// TIA Portal project "Project1" (V14)

(* hardware
DEVICE "S71500/ET200MP station_1"  S7-1500 station
   slot 0: "Rail_0"  Rack  6ES7 590-1***0-0AA0
   slot 1: "SERVER_PID"  CPU 1512C-1 PN  6ES7 512-1CK00-0AB0  V2.1
      slot 3: "CPU display_1"  6ES7591-1AA00-0AA0
*)

// ===== PLC "SERVER_PID"  CPU 1512C-1 PN =====

VAR_GLOBAL   // PLC tag table "Default tag table"
   ""Temperature_input"" AT %IW0 : Word;
   ""Pump_out"" AT %QW0 : Word;
END_VAR